(* PLC project x *)

PROGRAM FBD_A
  VAR
    tmr : TON;
  END_VAR
  VAR  (* added by the conversion: wires and edge detectors of the diagram *)
    _ADD24_ENO : BOOL;
    _ADD24_OUT : ANY;
  END_VAR

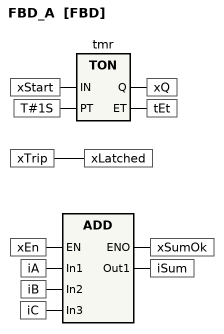
(* FBD diagram, written out as Structured Text *)
tmr(IN := xStart, PT := T#1S);
xQ := tmr.Q;
tEt := tmr.ET;
IF xTrip THEN xLatched := TRUE; END_IF;
_ADD24_OUT := ADD(EN := xEn, IN1 := iA, IN2 := iB, IN3 := iC, ENO => _ADD24_ENO);
IF _ADD24_ENO THEN iSum := _ADD24_OUT; END_IF;
xSumOk := _ADD24_ENO;
END_PROGRAM
